// TIA Portal V19 export
FUNCTION "FC_WT_from_Pos" : Void   // FC57, STL
TITLE = Umladen eines Wt aus einer Pos an FW/QT
{ S7_Optimized_Access := 'FALSE' }
// Aufruf aus FW bzw. QT
// stored: AutoNumber false
   VAR_INPUT
      Pos_Nr : USInt;
      send_DBEvt : Bool;   // Datenbank-Events senden
   END_VAR
   VAR_OUTPUT
      load_ok : Bool;
   END_VAR
   VAR_IN_OUT
      WT_Nr : Byte;
      WT_Nr_lang : DWord;
   END_VAR
   VAR_TEMP
      not_load : Bool;
      WT_DB : Word;
      Param : DWord;
      MW_Strom : Real;
      MD_Nr : USInt;
      inf_1 : Byte;
   END_VAR
BEGIN

NETWORK
TITLE = 
//----------------------------
//laden der Pos und prüfen
//----------------------------
      SET;
      R     #load_ok;

      CALL  "FC_POS_TO_WORK"
      ( Akt_Pos  := #Pos_Nr,
        not_load := #not_load
      );

      A     #not_load;
      BEC;

      L     0;
      L     "DB_POS".POS[0].WT_DB;
      >=I;
      BEC;

//----------------------------
//Umladen erlaubt
//----------------------------
      S     #load_ok;
      T     #WT_Nr;
      L     100;
      +I;
      T     #WT_DB;

      L     "DB_POS".POS[0].WT_Nr_lang;
      T     #WT_Nr_lang;

//----------------------------
//Abbruch --> Restzeit sichern
//----------------------------
      AN    "DB_POS".POS[0].ignor_Exp;
      L     0;
      JC    noZw;
      L     "DB_POS".POS[0].Restzeit;
noZw: OPN   DB [#WT_DB];
      L     %DBD50;  //Sicherung der fehlenden Expozeit am WT
      +D;
      T     %DBD50;  //Sicherung der fehlenden Expozeit am WT

      AN    #send_DBEvt;
      JC    noDB;

//----------------------------
//WT in Pos löschen
//----------------------------
noDB: L     0;
      T     "DB_POS".POS[0].WT_DB;  //WT_Nr_Kurz im Bad
      T     "DB_POS".POS[0].WT_Nr_lang;  //WT_Nr lang im Bad

//----------------------------
//Position aktualisieren
//----------------------------
      CALL  "FC_Pos_Behandlung"
      ( Pos_Nr     := #Pos_Nr,
        send_DBEvt := #send_DBEvt
      );
//-------------------------------
//zurückladen der PosDaten
//-------------------------------
      CALL  "FC_WORK_TO_POS"
      ( Akt_Pos := #Pos_Nr
      );

END_FUNCTION
